TYPE OperatingModeHomeing :
STRUCT
	PreconditionsFullfilled	:	BOOL;
	IsActive	:	BOOL;
	IsReached	:	BOOL;
	AllMachinesInHome	:	BOOL;
END_STRUCT
END_TYPE

(* stored: Version 1.1.0.1
   DUT OperatingModeHomeing: Id {dd0e6127-1187-4e5a-bb52-77fa0617157b} *)
